FUNCTION_BLOCK FB_BottomMold
VAR CONSTANT
	sCycleStateTextDef: ARRAY[0..30]  OF STRING :=	
		['State 0: Wait for Start',
		'State 1: Wait for transfer / drying ready to move in',
		'State 2: Move bottom mold in',
		'State 3: Move take out vertical up',
		'State 4: Move take out vertical down',
		'State 5: Wait for transfer is down, and vacuum on',
		'State 6: Move out, Move take out unit to out position',
		'State 7: Wait for product is picked up by gantry',
		'State 8: Move take out unit in',
		'State 9: Spare',
		'State 10: Spare',
		'State 11: Spare',
		'State 12: Spare',
		'State 13: Spare',
		'State 14: Spare',
		'State 15: Spare',
		'State 16: Spare',
		'State 17: Spare',
		'State 18: Spare',
		'State 19: Spare',
		'State 20: [Paused] wait for start',
		'State 21: Spare',
		'State 22: Spare',
		'State 23: Spare',
		'State 24: Spare',
		'State 25: StopDirect',
		'State 26: Error'];
	
	tCycleStateTimeouts: ARRAY[0..10] OF TIME := 
		[T#10S,T#10S,T#10S,T#10S,T#10S,T#10S,T#10S,T#10S,T#10S,T#10S,
		T#10S];

	sInitStateTextDef: ARRAY[0..10] OF STRING :=
		['State 0: Wait for Init start',
		'State 1: Move vertical air cylinder down',
		'State 2: Move bottommold out',
		'State 3; Move horizontal air cylinder out',
		'State 4: ',
		'State 5: ',
		'State 6: ',
		'State 7: ',
		'State 8: ',
		'State 9: ',
		'State 10: Stop init state'];

	tInitStateTimeouts: ARRAY[0..10] OF TIME := 
		[T#10S,T#10S,T#10S,T#10S,T#10S,T#10S,T#10S,T#10S,T#10S,T#10S
		,T#10S];
END_VAR

VAR_INPUT
	mxResetCycleState				: BOOL;
	mxResetInitState				: BOOL;
	mxForceInit						: BOOL; (*Reset Calibration Flag*)
	mxReset							: BOOL;	(*Reset Error*)
	mxEmergency						: BOOL;
	mxDoorsOpened					: BOOL;
	mxAutoMode						: BOOL; (* TRUE = Automode *)
	mxEmptyMachine					: BOOL;
	mxEnableHeating					: BOOL;



	mxGantryPickedUpProduct			: BOOL;

	mxTransferIsAtTransferPos		: BOOL;
	TransferPosA					: REAL;
	TransferPosB					: REAL;
	ContinueWithA					: BOOL;
	ContinueWithB					: BOOL;

	mxProductReadyForGantry			: BOOL; (* Signal to gantry, take out product *)


	mxVacuumOn						: BOOL;
	mxProductOnTopMold				: BOOL;

	ActualPositionTransfermold		: REAL;
	RHSR_Blocked 					: BOOL;
	
	(*Signals*)
	SgMoveIn						: BOOL; (* Signal from transfer mold *)
	sgMoveOut						: BOOL; (* Signal from transfer mold *)
	SgBottomIsIn					: BOOL; (* Signal to transfer *)
	SgBottomIsOut					: BOOL; (* Signal to TopMold, move down to dry *)
	SgMoldsAreClosed				: BOOL; (* Signal that indicates that the topmold is closed on the bottommold.*)
	sgEmptying						: BOOL; // machine is emptying.
	sgSample						: BOOL; // Block vacuum when bottommold goes in (Sample has been taken out).
	
	SgElapsedDryingTime				: TIME;
	SgTotalDryingTime				: TIME;
	
	sgTopmoldBlowOffReady			: BOOl; (*Signal from the topmold, the takeout may depart.*)
END_VAR
VAR_IN_OUT
	MachParameters					: ST_BottomMoldMachPar;
	SysParameters					: ST_BottomMoldSysPar;
	ProdParameters					: ST_BottomMoldProdPar;
END_VAR
VAR_OUTPUT
(*Errors*)
	Errors							: ST_BottomMoldErrors;
	mxErrorInit						: BOOL;		(* Error, stop immediately. Initialisation neccesary *)
	mxErrorStopinPos				: BOOL;		(* Error, stop in position. Only reset neccesary *)

(* State vars *)
	mxCycleBusy						: BOOL;
	mxInitBusy						: BOOL;
	
(* Vars *)
	mxInitialized					: BOOL;
	mxReadyForTransfer				: BOOL;
		
	mxProductReadyAtTakeOut			: BOOL; (* Signal to gantry, take out product *)
	mxTakeoutIsMovingUp				: BOOL;
	sgTakeOutUnitDown				: BOOL;
	
	mxCilIsMovingIn					: BOOL;
	mxCilIsMovingOut				: BOOL;
	mxCilIsIn						: BOOL;
	mxCilIsOut						: BOOL;	
	mxHorCilIsIn					: BOOL;
	mxHorCilIsOut					: BOOL;
	mxVertCilIsIn					: BOOL;
	mxVertCilIsOut					: BOOL;
	
	ActualPosition					: REAL;
END_VAR
VAR
(* State vars *)
	miCycleState					: INT :=0;
	miCycleOldstate					: INT :=0;
	mxCycleTransitionState			: BOOL := FALSE;
	sCycleStateText					: STRING;
	exCycleTimeOut					: BOOL;		(* Timeout for the whole programcycle *)
	CycleTimeout					: TON;
	CycleTimeOutUpFlank				: R_TRIG;
	mxCycleTimeoutEnable			: BOOL;
	CycleTime						: REAL;
	mxCycleHasError					: BOOL;
	miStopState						: INT;
	mxStartCycle					: BOOL;
	mxStopCycle						: BOOL;
	mxStopDirect					: BOOL;
	
	miInitState						: INT	:=0;
	miInitOldstate					: INT	:=0;
	mxInitTransitionState			: BOOL	:= FALSE;
	sInitStateText					: STRING;
	exInitTimeOut					: BOOL;		(* Timeout for the whole programcycle *)
	InitTimeout						: TON;
	InitTimeOutUpFlank				: R_TRIG;
	mxInitTimeoutEnable				: BOOL;
	InitTime						: REAL;
	mxInitHasError					: BOOL;
	mxStartInit						: BOOL;
	mxStopInit						: BOOL;
	

(* Objects *)
	HorizontalCilinder				: FB_BiValve2Fdbck;
	VerticalCilinder				: FB_BiValve2Fdbck;
	HorizontalAxis					: FB_NcAxis;
	VacuumTakeout					: ARRAY [1..6] OF FB_MonoValveNoFdbck;	(* IMD-V *)		
	VacuumSensor					AT %I* : ARRAY [1..6] OF BOOL;
	
	HeatingZone						: ARRAY [1..6] OF FB_Heatingzone;
	

	Vacuum							: FB_MonoValveNoFdbck;	(* IMD-V *)		
	BlowOff							: FB_MonoValveNoFdBck;
	
(* Vars *)
	T_TakeOutTime					: TON;
	T_VacSectionDelay				: ARRAY [1..6] OF TON;
	SR_ErrorNoVacAtSection			: ARRAY [1..GVL.MaxNrOfVacSectTakeOutUnit] OF SR;
	mxSwitchVacuumOn				: BOOL;
	miVacSection					: INT;
	T_VCilinderMoveOut				: TON;
	T_VCilinderMoveIn				: TON;
	
	RT_GantryPickedUpProduct 		: R_TRIG;
	//T_VacuumDelayedOff				: TON;
	FT_SwitchVacuumOff				: F_TRIG;
	T_TestBigBang					: TON;
	mxFirstCycle					: BOOL;
	
	mrAxisIsMoving					: BOOL;
	mrAxisActPos					: LREAL;
	RT_MoveToGreasingPosition: R_TRIG;
	mxHMI_MoveToGreasingPos: BOOL;
	T_VacuumBottomMoldClosed: TON;
	RT_VacuumBottomMoldClosed: R_TRIG;
	mxInPause: BOOL;
	RT_BlowOff: R_TRIG;
	T_BlowoffTime: TON;
	T_KickOffs: TON;
	NrOfKickoffs: REAL;
	mxResetBotStroke: BOOL;
END_VAR

Error();
Init();
Cycle();
Objects();

ActualPosition := LREAL_TO_REAL(HorizontalAxis.ActPosition);

mxCilIsIn := ((ActualPosition < (MachParameters.PositionInStop + 1)) AND (ActualPosition > (MachParameters.PositionInStop - 1))); 
mxCilIsOut := ((ActualPosition < (MachParameters.PositionOutStop + 1)) AND (ActualPosition > (MachParameters.PositionOutStop - 1))); 

mxCilIsMovingIn := HorizontalAxis.mxAxisIsMoving AND HorizontalAxis.axAxis.Status.NegativeDirection;
mxCilIsMovingOut := HorizontalAxis.mxAxisIsMoving AND HorizontalAxis.axAxis.Status.PositiveDirection;

// Move to Greasing Position
IF mxHMI_MoveToGreasingPos AND NOT mxCycleBusy AND NOT mxAutoMode THEN
	IF HorizontalAxis.M_MoveAbsolute(MachParameters.GreasingVelocity, MachParameters.GreasingPosition) THEN
		mxHMI_MoveToGreasingPos := FALSE;
	END_IF	
END_IF

IF mxResetBotStroke THEN
	mxResetBotStroke := FALSE;
	MachParameters.KickOffCounter :=0;
END_IF

ACTION Cycle:
(*StateChange (Transition)  Signalgeneration*)
mxCycleTransitionState:=(miCycleState<>miCycleOldstate);
(*State text*)
sCycleStateText:=sCycleStateTextDef[miCycleState];
(*Timeout Watchdog for Statemachine*)
mxCycleTimeoutEnable:=NOT (miCycleState=0) AND NOT mxReset;

CycleTimeout(IN:=mxCycleTimeoutEnable, PT:=tCycleStateTimeouts[miCycleState] );
CycleTimeOutUpFlank(CLK:=CycleTimeout.Q );
miCycleOldstate:=miCycleState;

(*Set Errorbit when Raising edge of Timeout has been detected*)
IF CycleTimeOutUpFlank.Q THEN
	exCycleTimeOut:=TRUE; 			(* 1 Timeout for the whole programcycle *)
END_IF

(*Function to reset the Statemachine*)
IF mxResetCycleState THEN
	mxResetCycleState:= FALSE;
	mxInitialized:= FALSE;
	miCycleState:=0;
	miCycleOldstate:=miCycleState;
	mxCycleTransitionState:=FALSE;

	mxStartCycle:= FALSE;
	mxStopCycle:= FALSE;
	mxStopDirect:= FALSE;
	mxTakeoutIsMovingUp:= FALSE; 
	mxProductReadyAtTakeOut:= FALSE;
	mxSwitchVacuumOn:= FALSE;
	SgBottomIsIn := FALSE;
	SgBottomIsOut := FALSE;
	sgMoveIn := FALSE;
	sgMoveOut := FALSE;
	sgTakeOutUnitDown := FALSE;
	mxEmptyMachine := FALSE;
	mxProductOnTopMold:= FALSE;
	T_VCilinderMoveIn.IN :=FALSE;
	HorizontalAxis.M_Stop();
	T_BlowOffTime.IN:=FALSE;
	BlowOff.M_Off();
	NrOfKickoffs := 0;
	T_KickOffs.IN := FALSE;
	
END_IF

(*Definition State has Error*)
mxCycleHasError:=FALSE;

T_KickOffs(IN:=, PT:=T#600S);
T_TakeOutTime(IN:=, PT:= MachParameters.VerticalCilinderTakeOutTime);
T_VCilinderMoveOut(IN:=, PT:= T#3S);
T_VCilinderMoveIn(IN:=, PT:=MachParameters.VerticalCilinderUpDelay);
T_VacuumBottomMoldClosed(IN:=, PT:=MachParameters.BottomMoldVacuumClosed);
RT_VacuumBottomMoldClosed(CLK:= MachParameters.ClosedVacEnabled AND SgMoldsAreClosed);
FT_SwitchVacuumOff(CLK:=mxSwitchVacuumOn);

IF RT_VacuumBottomMoldClosed.Q THEN
	T_VacuumBottomMoldClosed.IN:=TRUE;
	Vacuum.M_On();
END_IF

IF T_VacuumBottomMoldClosed.Q THEN
	T_VacuumBottomMoldClosed.IN:=FALSE;
	Vacuum.M_Off();
END_IF

//Gantry picked up product from the Takeout unit 
RT_GantryPickedUpProduct(CLK:= mxGantryPickedUpProduct);

IF mxSwitchVacuumOn AND mxAutoMode THEN
	IF MachParameters.EnableVacuumSection[1] THEN VacuumTakeout[1].M_On(); END_IF
	IF MachParameters.EnableVacuumSection[2] THEN VacuumTakeout[2].M_On(); END_IF
	IF MachParameters.EnableVacuumSection[3] THEN VacuumTakeout[3].M_On(); END_IF
	IF MachParameters.EnableVacuumSection[4] THEN VacuumTakeout[4].M_On(); END_IF
END_IF 

IF FT_SwitchVacuumOff.Q AND mxAutoMode THEN
	IF MachParameters.EnableVacuumSection[1] THEN VacuumTakeout[1].M_Off(); END_IF
	IF MachParameters.EnableVacuumSection[2] THEN VacuumTakeout[2].M_Off(); END_IF
	IF MachParameters.EnableVacuumSection[3] THEN VacuumTakeout[3].M_Off(); END_IF
	IF MachParameters.EnableVacuumSection[4] THEN VacuumTakeout[4].M_Off(); END_IF
END_IF

IF (miCycleState >= 3 AND miCycleState <= 5) AND NOT sgSample THEN	
		IF (ContinueWithA AND (ActualPositionTransfermold < (TransferPosA + MachParameters.StartVacAtTrPosOffset))) OR // At an ofset of transfermold pos
		 (ContinueWithB AND (ActualPositionTransfermold < (TransferPosB + MachParameters.StartVacAtTrPosOffset))) THEN	// Open the vacuum valve.
			Vacuum.M_On();
		END_IF
END_IF

RT_BlowOff(CLK:=SgElapsedDryingTime > (SgTotalDryingTime - MachParameters.OffsetStartBlowOff));
T_BlowoffTime(IN:=, PT:=MachParameters.BlowOffTime);


IF RT_BlowOff.Q THEN
	T_BlowoffTime.IN:=TRUE;
	BlowOff.M_On();
END_IF

IF T_BlowoffTime.Q THEN
	T_BlowOffTime.IN:=FALSE;
	BlowOff.M_Off();
END_IF

(*Cycle State's*)
CASE miCycleState OF

	0:  // (P)  Wait for start 
		IF mxStopCycle THEN
			mxStopCycle:= FALSE;
			miStopState:= miCycleState;
			miCycleState:= 20;
		ELSIF mxStartCycle THEN
			mxStartCycle:= FALSE;
			miCycleState:= 1;
		END_IF	

	1:  // (P)  Wait for transfer/Drying ready to move in 
		IF mxStopDirect THEN
			mxStopDirect:= FALSE;
			miCycleState:= 25;
		ELSIF mxStopCycle AND mxEmptyMachine THEN
			mxStopCycle:=False;
			mxEmptyMachine:= FALSE;
			miCycleState:= 0;
		ELSIF mxStopCycle THEN
			mxStopCycle:= FALSE;
			miStopState:= miCycleState;
			miCycleState:= 20;
		ELSIF SgMoveIn THEN
			SgMoveIn:= FALSE;
			SgBottomIsOut:= FALSE;
			
			T_KickOffs.IN := TRUE;
			miCycleState:= 2;
		END_IF

	2:	// (NP) Move IN
		IF mxStopDirect THEN
			mxStopDirect:= FALSE;
			miCycleState:= 25;
		ELSIF HorizontalAxis.M_MoveAbsolute(MachParameters.AxisVelocityAuto, MachParameters.PositionInStop) AND HorizontalCilinder.M_In() THEN
			SgBottomIsIn:= TRUE;
			SgBottomIsOut := FALSE;
			MachParameters.KickOffCounter := MachParameters.KickOffCounter +1;
			miCycleState:=3;
		END_IF

	3:	// (P) Move Take out vertical Up (bateu: changed NP to P -> 20190408)
		IF mxStopDirect THEN
			mxStopDirect:= FALSE;
			miCycleState:= 25;
		ELSIF mxStopCycle THEN
			mxStopCycle:= FALSE;
			miStopState:= miCycleState;
			mxSwitchVacuumOn:= FALSE;		// Close vacuum valve if it was opened allready	
			Vacuum.M_Off();					// Close vacuum of bottommold (starts at top off cycle).
			miCycleState:= 20;
		ELSIF mxProductOnTopMold THEN									// check if there is a product				
			IF (VerticalCilinder.M_In_Pressure()) THEN //OR T_VCilinderMoveIn.Q) THEN	// if there is a product, Get it with the cylinder. //MZE 20190404 Replaced method M_In				
				mxTakeoutIsMovingUp:= TRUE;								// when cilinder is up signal topmold to start blowoff
				mxSwitchVacuumOn:= TRUE;
				IF sgTopmoldBlowOffReady THEN
					miCycleState:= 4;
				END_IF
			END_IF
		ELSE 
			miCycleState:= 5;
		END_IF

	4:	// (NP) Move take out vertical down 	
		T_TakeOutTime.IN:= TRUE;
		mxTakeoutIsMovingUp:= FALSE;		
		IF mxStopDirect THEN
			mxStopDirect:= FALSE;		
			miCycleState:= 25;
		ELSIF TRUE THEN		
			IF VerticalCilinder.M_Out() THEN
				sgTakeOutUnitDown := TRUE;
				T_TakeOutTime.IN:= FALSE;
				IF NOT mxEmptyMachine THEN
					miCycleState:= 5;
				ELSE
					miCycleState:= 6;
				END_IF
			END_IF
		END_IF		

	5:  // (P)  Wait for transfer is down, vacuum on
		IF mxStopDirect THEN
			mxStopDirect:= FALSE;
			miCycleState:= 25;
		ELSIF mxStopCycle THEN
			mxStopCycle:= FALSE;
			miStopState:= miCycleState;
			Vacuum.M_Off(); 	// gets restarted above cycle.
			miCycleState:= 20;
		ELSIF sgMoveOut THEN	// When the closed wait time has elapsed and tranfer is up.
			sgMoveOut:= FALSE;
			miCycleState:= 6;
		END_IF
		
	6:  // (NP) Move OUT, takeout horizontal out
		IF HorizontalAxis.ActPosition > (MachParameters.PositionOutStop - MachParameters.StopVacAtBmPosOffset) THEN
			Vacuum.M_Off();
		END_IF
		
		IF HorizontalAxis.ActPosition > (MachParameters.PositionOutStop - MachParameters.StartVacBeforeDryingAtBmPosOffset) AND NOT sgSample AND NOT sgEmptying THEN
			Vacuum.M_On();
		END_IF
		
		IF mxStopDirect THEN
			mxStopDirect:= FALSE;	
			miCycleState:= 25;
		ELSIF HorizontalAxis.M_MoveAbsolute(MachParameters.AxisVelocityAuto,MachParameters.PositionOutStop) AND HorizontalCilinder.M_Out() THEN
			sgTakeOutUnitDown := FALSE;
			SgBottomIsOut:= TRUE;
			SgBottomIsIn:= FALSE;
			mxSwitchVacuumOn:= FALSE;
			MachParameters.KickOffCounter := MachParameters.KickOffCounter +1;			
			IF mxProductOnTopMold THEN mxProductReadyAtTakeOut:= TRUE; END_IF
			miCycleState:= 7;
		END_IF

	7:	// (P)  Wait for product is picked up by gantry	
		IF mxStopDirect THEN
			mxStopDirect:= FALSE;
			miCycleState:= 25;
		ELSIF mxStopCycle THEN
			mxStopCycle:= FALSE;
			miStopState:= miCycleState;
			mxProductReadyAtTakeOut:=FALSE; // Set this false because gantry expects a pulse.
			miCycleState:= 20;
		ELSIF (mxProductOnTopMold AND RT_GantryPickedUpProduct.Q) OR NOT mxProductOnTopMold THEN
			mxProductReadyAtTakeOut := FALSE; // -> stop signaling the gantry that there is a product ready to take
			mxProductOnTopMold:= FALSE;
			mxGantryPickedUpProduct:= FALSE;
			miCycleState:= 8;
		END_IF

	8: 	// (NP) Move Takeout IN 
		IF mxStopDirect THEN
			mxStopDirect:= FALSE;		
			miCycleState:= 25;
		ELSIF HorizontalCilinder.M_In() THEN
			NrOfKickoffs := TIME_TO_REAL(T_KickOffs.ET);	// Calculate the time this run took.
			T_KickOffs.IN := FALSE;	
			
			miCycleState:= 1;
		END_IF

	20:	// Pause state
		NrOfKickoffs := 0;
		T_KickOffs.IN := FALSE;
	
		
		
		IF mxStopDirect THEN
			mxStopDirect:= FALSE;
			miCycleState:= 25;
		ELSIF mxStartCycle THEN
			IF miStopState = 7 AND mxProductOnTopMold THEN
				mxProductReadyAtTakeOut := mxProductOnTopMold; // resignal gantry to get product from takeout unit.
			END_IF

			mxStartCycle:= FALSE;
			miCycleState:= miStopState;			
		END_IF

	25: // Stop Direct 
		mxInitialized:= FALSE;

		mxStartCycle:= FALSE;
		mxStopCycle:= FALSE;
		mxStopDirect:= FALSE;
		
		mxTakeoutIsMovingUp:= FALSE; 
		mxSwitchVacuumOn:= FALSE;
		SgBottomIsIn := FALSE;
		SgBottomIsOut := FALSE;
		sgMoveIn := FALSE;
		sgMoveOut := FALSE;
		sgTakeOutUnitDown := FALSE;
		
		HorizontalAxis.M_Stop();
		
		Vacuum.M_Off();
		T_BlowOffTime.IN:=FALSE;
		BlowOff.M_Off();
	
		NrOfKickoffs := 0;
		T_KickOffs.IN := FALSE;		

		miCycleState:= 0;
END_CASE

mxCycleBusy:= miCycleState<>0 AND NOT (miCycleState=20);
mxInPause:=miCycleState=20;
END_ACTION

ACTION Error:
T_VacSectionDelay[1](PT:= T#3S);
T_VacSectionDelay[2](PT:= T#3S);
T_VacSectionDelay[3](PT:= T#3S);
T_VacSectionDelay[4](PT:= T#3S);
T_VacSectionDelay[5](PT:= T#3S);
T_VacSectionDelay[6](PT:= T#3S);

FOR miVacSection:= 1 TO GVL.MaxNrOfVacSectTakeOutUnit DO
	T_VacSectionDelay[miVacSection].IN:= VacuumTakeout[miVacSection].mxIsOn;
	SR_ErrorNoVacAtSection[miVacSection](SET1:= MachParameters.EnableVacuumSection[miVacSection] AND VacuumTakeout[miVacSection].mxIsOn AND 
	(T_VacSectionDelay[miVacSection].Q AND NOT VacuumSensor[miVacSection]), 
	RESET:= mxReset, Q1=> Errors.VacuumSection[miVacSection]);
END_FOR

(*************************************************************************************************)
mxErrorStopinPos:= FALSE;
mxErrorInit:=HorizontalAxis.ErrorStop OR HorizontalCilinder.mxErrorInit  OR VerticalCilinder.mxErrorInit 
			OR HeatingZone[1].mxErrorInit
			OR HeatingZone[2].mxErrorInit
			OR HeatingZone[3].mxErrorInit
			OR HeatingZone[4].mxErrorInit
			OR HeatingZone[5].mxErrorInit
			OR HEatingZone[6].mxErrorInit;
END_ACTION

ACTION Init:
(*StateChange (Transition)  Signalgeneration*)
mxInitTransitionState:=(miInitState<>miInitOldstate);
(*State text*)
sInitStateText:=sInitStateTextDef[miInitState];
(*Timeout Watchdog for Statemachine*)
mxInitTimeoutEnable:=NOT (miInitState=0)  AND NOT mxReset;

InitTimeout(IN:=mxInitTimeoutEnable  , PT:=tInitStateTimeouts[miInitState] );
InitTimeOutUpFlank(CLK:=InitTimeout.Q );
miInitOldstate:=miInitState;

(*Set Errorbit when Raising edge of Timeout has been detected*)
IF InitTimeOutUpFlank.Q THEN
	exInitTimeOut:=TRUE; 			(* 1 Timeout for the whole programcycle *)
END_IF

(*Function to reset the Statemachine*)
IF mxResetInitState THEN
	mxResetInitState:=FALSE;
	miInitState:=0;
	miInitOldstate:=miInitState;
	mxInitTransitionState:=FALSE;

	mxStartInit:= FALSE;
	mxStopInit:= FALSE;
	
END_IF

(*Definition State has Error*)
mxInitHasError:=FALSE;

(*Init State's*)
CASE miInitState OF
	0:
		IF mxStartInit THEN
			mxStartInit:= FALSE;
			mxInitialized:= FALSE;
			Vacuum.M_Off();
			mxSwitchVacuumOn:= FALSE;
			
			miInitState:= 1;
		END_IF

	(* Vertical cilinder Down *)
	1:
		IF mxStopInit THEN
			mxStopInit:= FALSE;
			
			miInitState:= 10;
		ELSIF VerticalCilinder.M_Out() THEN	(*BaTeu, changed M_in to M_out (In = Up / out = down) *)
			
			miInitState:= 2;
		END_IF
	
	(* Move OUT *)
	2:
		IF mxStopInit THEN
			mxStopInit:= FALSE;
			
			miInitState:= 10;
		ELSIF HorizontalAxis.M_MoveAbsolute(MAchparameters.AxisVelocityInit, MachParameters.PositionOutStop) THEN

			miInitState:= 3;
		END_IF

	(* Horizontal cilinder Out *)
	3:
		IF mxStopInit THEN
			mxStopInit:= FALSE;
			
			miInitState:= 10;
		ELSIF HorizontalCilinder.M_Out() THEN

			mxInitialized:= TRUE;
			miInitState :=0;
		END_IF	

	(* Stop Init *)
	10:
		HorizontalAxis.M_Stop();
		mxStartInit:= FALSE;
		mxStopInit:= FALSE;
		mxInitialized:= FALSE;
		
		miInitState:= 0;
			
END_CASE

mxInitBusy:= miInitState<>0;
END_ACTION

METHOD M_EmptyMachine

IF mxCycleBusy THEN
	mxEmptyMachine:= TRUE;	
END_IF
END_METHOD

METHOD M_StartCycle

IF NOT mxCycleBusy THEN
	mxStopCycle := FALSE;
	mxStartCycle:= TRUE;	
END_IF
END_METHOD

METHOD M_StartInit

IF NOT mxInitBusy THEN 
	mxStartInit:= TRUE; 
END_IF
END_METHOD

METHOD M_StopCycle
mxStopCycle:= TRUE;
END_METHOD

METHOD M_StopDirect

IF mxCycleBusy THEN
	mxStopDirect:= TRUE;	
END_IF
END_METHOD

METHOD M_StopInit

IF mxInitBusy THEN 
	mxStopInit:= TRUE; 
END_IF
END_METHOD

ACTION Objects:
HorizontalAxis(
	mxEnable:= NOT mxEmergency OR NOT mxDoorsOpened, 
	mxInhibit:= RHSR_Blocked, //20190124 (was hard FALSE).
	mxAutoMode:= mxAutoMode, 
	mxReset:= mxReset, 
	mxFirstCycle:= mxFirstCycle, 
	mxEmergency:= mxEmergency, 
	mxSimulation:= , 
	mxResetCycle:= , 
	mxDisable_Positive:= FALSE,
	mxDisable_Negative:= FALSE,
	mxBlockHMI:= , 
	mrOverride:=100.0 , 
	mrVelocityManual:= MachParameters.AxisVelocityManual,  
	mrHomePos:= MachParameters.AxisPositionHome, 
	SysParameters:= SysParameters.BottomMoldAxis,
	mxAxisIsMoving=> mrAxisIsMoving, 
	Errors=> Errors.HorizontalAxis, 
	ActPosition=>mrAxisActPos );
	
Vacuum(
	mxReset:= mxReset, 
	mxEmergency:= mxEmergency OR mxDoorsOpened, 
	mxAutoMode:= mxAutoMode);

VacuumTakeout[1](
	mxReset:=mxReset , 
	mxEmergency:= mxEmergency OR mxDoorsOpened, 
	mxAutoMode:=mxAutoMode , 
	mxIsOn=>);

VacuumTakeout[2](
	mxReset:=mxReset , 
	mxEmergency:= mxEmergency OR mxDoorsOpened, 
	mxAutoMode:=mxAutoMode , 
	mxIsOn=>);
	
VacuumTakeout[3](
	mxReset:=mxReset , 
	mxEmergency:= mxEmergency OR mxDoorsOpened, 
	mxAutoMode:=mxAutoMode , 
	mxIsOn=>);
	
VacuumTakeout[4](
	mxReset:=mxReset , 
	mxEmergency:= mxEmergency OR mxDoorsOpened, 
	mxAutoMode:=mxAutoMode , 
	mxIsOn=>);
	
VacuumTakeout[5](
	mxReset:=mxReset , 
	mxEmergency:= mxEmergency OR mxDoorsOpened, 
	mxAutoMode:=mxAutoMode , 
	mxIsOn=>);	
	
VacuumTakeout[6](
	mxReset:=mxReset , 
	mxEmergency:= mxEmergency OR mxDoorsOpened, 
	mxAutoMode:=mxAutoMode , 
	mxIsOn=>);
		
(* Take out Unit *)
HorizontalCilinder(
	mxReset:= mxReset, 
	mxEmergency:=  mxEmergency OR mxDoorsOpened, 
	mxAutoMode:= mxAutoMode, 
	MachParameters:= MachParameters.HorizontalCilinder, 
	mxIsVertical:=FALSE,
	mxIsIn=> mxHorCilIsIn, 
	mxIsOut=> mxHorCilIsOut, 
	Errors=> Errors.HorizontalCilinder);
	
VerticalCilinder(
	mxReset:= mxReset, 
	mxEmergency:=  mxEmergency OR mxDoorsOpened, 
	mxAutoMode:= mxAutoMode, 
	MachParameters:= MachParameters.VerticalCilinder, 
	mxIsVertical:=TRUE,
	mxIsIn=> mxVertCilIsIn, 
	mxIsOut=> mxVertCilIsOut, 
	Errors=> Errors.VerticalCilinder);

HeatingZone[1](
	mxReset:= mxReset,
	mxEmergency:=mxEmergency OR mxDoorsOpened,
	mxDoorsOpened:=FALSE,
	mxEnableHeating:=mxEnableHeating,
	MachParameters:=MachParameters.HeatingZone[1],
	Errors=> Errors.HeatingZone[1]);

HeatingZone[2](
	mxReset:= mxReset,
	mxEmergency:=mxEmergency OR mxDoorsOpened,
	mxDoorsOpened:=FALSE,
	mxEnableHeating:=mxEnableHeating,
	MachParameters:=MachParameters.HeatingZone[2],
	Errors=> Errors.HeatingZone[2]);

HeatingZone[3](
	mxReset:= mxReset,
	mxEmergency:=mxEmergency OR mxDoorsOpened,
	mxDoorsOpened:=FALSE,
	mxEnableHeating:=mxEnableHeating,
	MachParameters:=MachParameters.HeatingZone[3],
	Errors=> Errors.HeatingZone[3]);

HeatingZone[4](
	mxReset:= mxReset,
	mxEmergency:=mxEmergency OR mxDoorsOpened,
	mxDoorsOpened:=FALSE,
	mxEnableHeating:=mxEnableHeating,
	MachParameters:=MachParameters.HeatingZone[4],
	Errors=> Errors.HeatingZone[4]);

HeatingZone[5](
	mxReset:= mxReset,
	mxEmergency:=mxEmergency OR mxDoorsOpened,
	mxDoorsOpened:=FALSE,
	mxEnableHeating:=mxEnableHeating,
	MachParameters:=MachParameters.HeatingZone[5],
	Errors=> Errors.HeatingZone[5]);

HeatingZone[6](
	mxReset:= mxReset,
	mxEmergency:=mxEmergency OR mxDoorsOpened,
	mxDoorsOpened:=FALSE,
	mxEnableHeating:=mxEnableHeating,
	MachParameters:=MachParameters.HeatingZone[6],
	Errors=> Errors.HeatingZone[6]);
END_ACTION

END_FUNCTION_BLOCK

(* stored: Version 1.1.0.1, ProductVersion 3.1.4020.12
   POU FB_BottomMold: Id {ccbf8089-291c-4aab-94f9-a44bd213a368}, SpecialFunc None
   Action Cycle: Id {ae3b5cab-4c78-4bb0-8feb-8ce871150b54}
   Action Error: Id {c4df5ba1-9a66-4098-86d4-b90ed497cf90}
   Action Init: Id {be5348c5-1e7b-4d14-8a83-11a73630b247}
   Method M_EmptyMachine: Id {8d25f409-41f7-42e5-a22e-e7a7df432e5b}
   Method M_StartCycle: Id {e67aad85-0604-47f1-ba47-55fa411ac9d5}
   Method M_StartInit: Id {b1603155-5875-4637-b9e7-7322b22e5028}
   Method M_StopCycle: Id {67078015-fce2-453c-bc24-705d492a5fa1}
   Method M_StopDirect: Id {3637dbb7-e0c0-400a-9a56-9c236c7a25f9}
   Method M_StopInit: Id {bddf29e3-2749-41e5-a185-d5ddaa20a853}
   Action Objects: Id {3dbdf37a-b6ab-487d-9bfd-5659ada96c89} *)
